Fanuc KAREL source: kb00088.KL

-- PROVISIONAL review KL for V940-1; original PC SHA256 f943db77a69e7230789e18694b47a4b4f91edb604577fb23cfd0f3b283e5894e
-- Incomplete behavior may be omitted. Consult companion uncertainty JSON. Do not deploy.
PROGRAM KB00088
%NOLOCKGROUP
BEGIN
  -- V9_ZERO_TABLE_METADATA_HINT layout=0002_ascii; no indexed target words; source/name/runtime held
  -- UNRESOLVED_PC offsets 5-12; opcodes 9D,23
  -- UNRESOLVED_PC offsets 17-24; opcodes 9D,23
  -- UNRESOLVED_PC offsets 29-36; opcodes 9D,23
  -- UNRESOLVED_PC offsets 41-77; opcodes 27,22,22,22,27,9D,31,7E,4A
  -- UNRESOLVED_PC offsets 82-86; opcodes 7F
END KB00088
